// TIA Portal V19 export
FUNCTION_BLOCK "DecoilersHRot_FB"   // FB40, LAD
TITLE = DECOILERS HORIZONTAL ROTATION
// stored: MemoryReserve 100, SetENOAutomatically false
   VAR_INPUT
      AreaInterface : "AreaInterface";
      ZSI : "udt_ZoneSafetyInterface";
      DSI : Struct
         Rotation : "udt_DeviceSafetyInterface";
         Pivot : "udt_DeviceSafetyInterface";
         Translation : "udt_DeviceSafetyInterface";
      END_STRUCT;
      Drive : Struct
         Traslation : "TAx_DriveInterface";
      END_STRUCT;
      HW_ID : Struct
         Traslation_TEL1 : HW_SUBMODULE;
         TraslationEnc_IO : HW_SUBMODULE;
      END_STRUCT;
      DataIn : Struct
         PB_Decoiler1_MoveInLine : Bool;
         PB_Decoiler2_MoveInLine : Bool;
         Rotation : "ValveMachine_DataIn";
         Pivot : "ValveMachine_DataIn";
         Traslation : "Positioning_DOL_Machine_DataIn";
      END_STRUCT;
      CIn : Struct
         Manager : "DecoilersHRot_Manager";
         CoilCar_OutOfLine : Bool;
         PressureRunning_Rotation : Bool;
         PressureRunning_Pivot : Bool;
      END_STRUCT;
      Config : Struct
         Rotation : "ValveMachine_Config";
         Pivot : "ValveMachine_Config";
         Traslation : "Positioning_DOL_Machine_Config";
      END_STRUCT;
   END_VAR
   VAR_OUTPUT
      MachineInterface : "MachineInterface";
      DataOut : Struct
         Rotation : "ValveMachine_DataOut";
         Pivot : "ValveMachine_DataOut";
         Tower_Lamp : Bool;
         Tower_Horn : Bool;
      END_STRUCT;
      COut : "DecoilersHRot_Status";
   END_VAR
   VAR_IN_OUT
      PersistentValues : Struct
         Par : Struct
            TraslationAx : "Positioning_DOL_Machine_Par";
            TraslationEnc : "PosFbk_RTN";
            Traslation_AutSpeed : Real;
         END_STRUCT;
         Ax_Pers : "Positioning_DOL_Machine_Pers_Data";
      END_STRUCT;
   END_VAR
   VAR
      Warning : Struct
         Rotation : "ValveMachine_Wng";
         Pivot : "ValveMachine_Wng";
         Traslation : "Positioning_DOL_Machine_Wng";
         Rotation_NotInPosition : Bool;
         Pivot_NotWork : Bool;
         Translation_NotInPosition : Bool;
      END_STRUCT;
      Alarm : Struct
         Rotation : "ValveAlr";
         Pivot : "ValveAlr";
         Traslation_Ax : "Positioning_DOL_Machine_Alr";
         Traslation_Enc : "PosFbk_Encoder_Alr";
         Rotation_NotInPosition : Bool;
         Pivot_NotWork : Bool;
      END_STRUCT;
      Sts : Struct
         Decoiler1_InLine_Partial : Bool;
         Decoiler2_InLine_Partial : Bool;
      END_STRUCT;
      Ctrl : Struct
         Decoiler1_MoveInLine_Man : Bool;
         Decoiler2_MoveInLine_Man : Bool;
         Decoiler1_MoveInLine_Aut : Bool;
         Decoiler2_MoveInLine_Aut : Bool;
         Decoiler1_MoveInLine : Bool;
         Decoiler2_MoveInLine : Bool;
      END_STRUCT;
      Rotation : "ValveMachine_FB";
      Pivot : "ValveMachine_FB";
      Translation : "Positioning_DOL_Machine_FB";
      Traslation_Enc : "PosFbk_SickAFM60";
      Traslation_EncITF : "PosFbk_ITF";
      TON_Rotation_NotInPosition : TON_TIME;
      TON_Pivot_NotWork : TON_TIME;
      TON_Translation_NotInPosition { S7_SetPoint := 'True'} : TON_TIME;
      AUX : Struct
         Move_Pb_InLineDecoiler1 : Bool;
         Move_Pb_InLineDecoiler2 : Bool;
      END_STRUCT;
   END_VAR
   VAR_TEMP
      Decoiler_N : Int;
      Target : LReal;
      InPosition : Bool;
   END_VAR
   VAR_TEMP   // added for the SCL form of the ladder/FBD networks
      _w1 : Bool;
      _w2 : Bool;
      _w3 : Bool;
   END_VAR
BEGIN

REGION Network 1: Man move in line
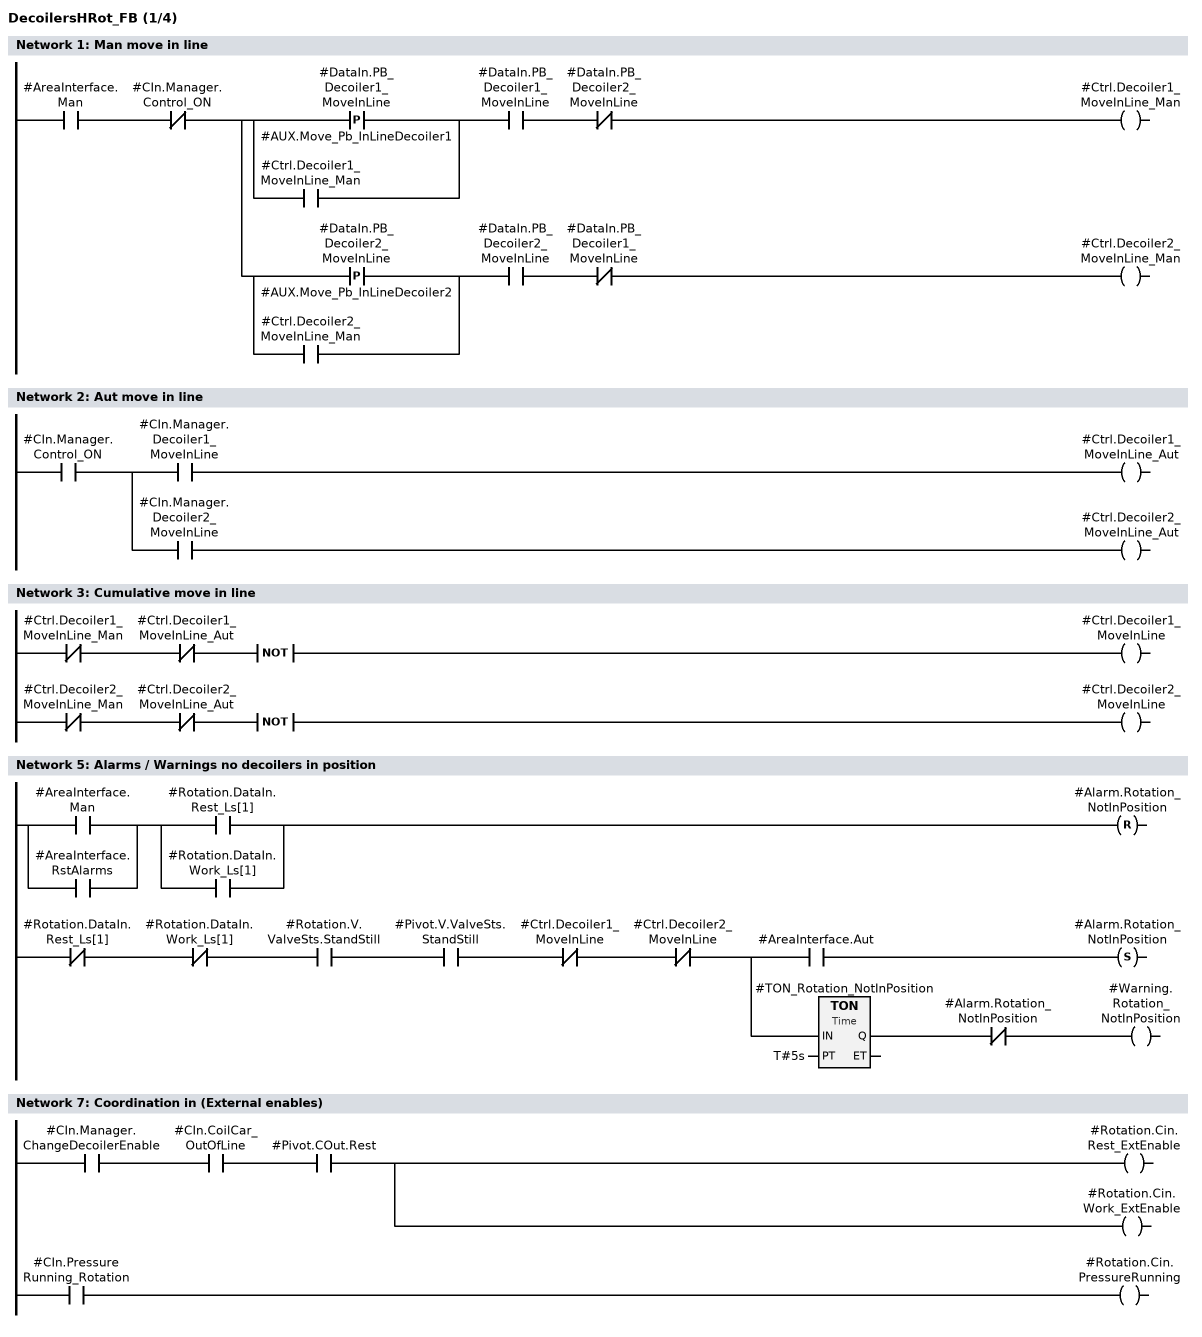
   RUNG wire#powerrail
      Contact( #AreaInterface.Man )
      I_Contact( #CIn.Manager.Control_ON )
      wire#w1
      P_Contact(operand := #DataIn.PB_Decoiler1_MoveInLine, bit := #AUX.Move_Pb_InLineDecoiler1)
      wire#w2
      Contact( #DataIn.PB_Decoiler1_MoveInLine )
      I_Contact( #DataIn.PB_Decoiler2_MoveInLine )
      Coil( #Ctrl.Decoiler1_MoveInLine_Man )
   END_RUNG
   RUNG wire#w1
      Contact( #Ctrl.Decoiler1_MoveInLine_Man )
   END_RUNG wire#w2
   RUNG wire#w1
      P_Contact(operand := #DataIn.PB_Decoiler2_MoveInLine, bit := #AUX.Move_Pb_InLineDecoiler2)
      wire#w3
      Contact( #DataIn.PB_Decoiler2_MoveInLine )
      I_Contact( #DataIn.PB_Decoiler1_MoveInLine )
      Coil( #Ctrl.Decoiler2_MoveInLine_Man )
   END_RUNG
   RUNG wire#w1
      Contact( #Ctrl.Decoiler2_MoveInLine_Man )
   END_RUNG wire#w3
   // the same network as SCL:
   #_w1 := #AreaInterface.Man AND NOT #CIn.Manager.Control_ON;
   #_w2 := #_w1 AND #DataIn.PB_Decoiler1_MoveInLine AND NOT #AUX.Move_Pb_InLineDecoiler1;   // rising edge of #DataIn.PB_Decoiler1_MoveInLine
   #AUX.Move_Pb_InLineDecoiler1 := #DataIn.PB_Decoiler1_MoveInLine;
   #Ctrl.Decoiler1_MoveInLine_Man := (#_w2 OR (#_w1 AND #Ctrl.Decoiler1_MoveInLine_Man)) AND #DataIn.PB_Decoiler1_MoveInLine AND NOT #DataIn.PB_Decoiler2_MoveInLine;
   #_w3 := #_w1 AND #DataIn.PB_Decoiler2_MoveInLine AND NOT #AUX.Move_Pb_InLineDecoiler2;   // rising edge of #DataIn.PB_Decoiler2_MoveInLine
   #AUX.Move_Pb_InLineDecoiler2 := #DataIn.PB_Decoiler2_MoveInLine;
   #Ctrl.Decoiler2_MoveInLine_Man := (#_w3 OR (#_w1 AND #Ctrl.Decoiler2_MoveInLine_Man)) AND #DataIn.PB_Decoiler2_MoveInLine AND NOT #DataIn.PB_Decoiler1_MoveInLine;
END_REGION

REGION Network 2: Aut move in line
   RUNG wire#powerrail
      Contact( #CIn.Manager.Control_ON )
      wire#w1
      Contact( #CIn.Manager.Decoiler1_MoveInLine )
      Coil( #Ctrl.Decoiler1_MoveInLine_Aut )
   END_RUNG
   RUNG wire#w1
      Contact( #CIn.Manager.Decoiler2_MoveInLine )
      Coil( #Ctrl.Decoiler2_MoveInLine_Aut )
   END_RUNG
   // the same network as SCL:
   #Ctrl.Decoiler1_MoveInLine_Aut := #CIn.Manager.Control_ON AND #CIn.Manager.Decoiler1_MoveInLine;
   #Ctrl.Decoiler2_MoveInLine_Aut := #CIn.Manager.Control_ON AND #CIn.Manager.Decoiler2_MoveInLine;
END_REGION

REGION Network 3: Cumulative move in line
   RUNG wire#powerrail
      I_Contact( #Ctrl.Decoiler1_MoveInLine_Man )
      I_Contact( #Ctrl.Decoiler1_MoveInLine_Aut )
      Not()
      Coil( #Ctrl.Decoiler1_MoveInLine )
   END_RUNG
   RUNG wire#powerrail
      I_Contact( #Ctrl.Decoiler2_MoveInLine_Man )
      I_Contact( #Ctrl.Decoiler2_MoveInLine_Aut )
      Not()
      Coil( #Ctrl.Decoiler2_MoveInLine )
   END_RUNG
   // the same network as SCL:
   #Ctrl.Decoiler1_MoveInLine := NOT (NOT #Ctrl.Decoiler1_MoveInLine_Man AND NOT #Ctrl.Decoiler1_MoveInLine_Aut);
   #Ctrl.Decoiler2_MoveInLine := NOT (NOT #Ctrl.Decoiler2_MoveInLine_Man AND NOT #Ctrl.Decoiler2_MoveInLine_Aut);
END_REGION

REGION Network 4: <<< ROTATION >>
END_REGION

REGION Network 5: Alarms / Warnings no decoilers in position
   RUNG wire#powerrail
      Contact( #AreaInterface.Man )
      wire#w1
      Contact( #Rotation.DataIn.Rest_Ls[1] )
      wire#w2
      R_Coil( #Alarm.Rotation_NotInPosition )
   END_RUNG
   RUNG wire#powerrail
      Contact( #AreaInterface.RstAlarms )
   END_RUNG wire#w1
   RUNG wire#w1
      Contact( #Rotation.DataIn.Work_Ls[1] )
   END_RUNG wire#w2
   RUNG wire#powerrail
      I_Contact( #Rotation.DataIn.Rest_Ls[1] )
      I_Contact( #Rotation.DataIn.Work_Ls[1] )
      Contact( #Rotation.V.ValveSts.StandStill )
      Contact( #Pivot.V.ValveSts.StandStill )
      I_Contact( #Ctrl.Decoiler1_MoveInLine )
      I_Contact( #Ctrl.Decoiler2_MoveInLine )
      wire#w3
      Contact( #AreaInterface.Aut )
      S_Coil( #Alarm.Rotation_NotInPosition )
   END_RUNG
   RUNG wire#w3
      { S7_Templates := "time_type := Time" } #TON_Rotation_NotInPosition.TON(pt := T#5s, et =>)
      I_Contact( #Alarm.Rotation_NotInPosition )
      Coil( #Warning.Rotation_NotInPosition )
   END_RUNG
   // the same network as SCL:
   IF (#AreaInterface.Man OR #AreaInterface.RstAlarms) AND (#Rotation.DataIn.Rest_Ls[1] OR #Rotation.DataIn.Work_Ls[1]) THEN
       #Alarm.Rotation_NotInPosition := FALSE;
   END_IF;
   #_w1 := NOT #Rotation.DataIn.Rest_Ls[1] AND NOT #Rotation.DataIn.Work_Ls[1] AND #Rotation.V.ValveSts.StandStill AND #Pivot.V.ValveSts.StandStill AND NOT #Ctrl.Decoiler1_MoveInLine AND NOT #Ctrl.Decoiler2_MoveInLine;
   IF #_w1 AND #AreaInterface.Aut THEN #Alarm.Rotation_NotInPosition := TRUE; END_IF;
   #TON_Rotation_NotInPosition(IN := #_w1, PT := T#5s);   // TON
   #Warning.Rotation_NotInPosition := #TON_Rotation_NotInPosition.Q AND NOT #Alarm.Rotation_NotInPosition;
END_REGION

REGION Network 6 (SCL): Coordination in (Manager)
   #Rotation.Cin.Manager.EnableStopDoorOpeningReq := #CIn.Manager.EnableStopDoorOpeningReq;
   #Rotation.Cin.Manager.EnableStopInPhase := #CIn.Manager.EnableStopInPhase;
   #Rotation.Cin.Manager.EnableStopProgrammed := #CIn.Manager.EnableStopProgrammed;

   // Rotazione @Rest = Decoiler 1 in linea
   // Rotazione @Work = Decoiler 2 in linea

   #Rotation.Cin.Manager.Rest := NOT #Rotation.COut.Rest AND #Ctrl.Decoiler1_MoveInLine;

   #Rotation.Cin.Manager.Work :=  NOT #Rotation.COut.Work AND #Ctrl.Decoiler2_MoveInLine;


   #Rotation.Cin.Manager.Control_ON := #CIn.Manager.Control_ON OR #Rotation.Cin.Manager.Rest OR #Rotation.Cin.Manager.Work;
END_REGION

REGION Network 7: Coordination in (External enables)
   RUNG wire#powerrail
      Contact( #CIn.Manager.ChangeDecoilerEnable )
      Contact( #CIn.CoilCar_OutOfLine )
      Contact( #Pivot.COut.Rest )
      wire#w1
      Coil( #Rotation.Cin.Rest_ExtEnable )
   END_RUNG
   RUNG wire#w1
      Coil( #Rotation.Cin.Work_ExtEnable )
   END_RUNG
   RUNG wire#powerrail
      Contact( #CIn.PressureRunning_Rotation )
      Coil( #Rotation.Cin.PressureRunning )
   END_RUNG
   // the same network as SCL:
   #Rotation.Cin.Rest_ExtEnable := #CIn.Manager.ChangeDecoilerEnable AND #CIn.CoilCar_OutOfLine AND #Pivot.COut.Rest;
   #Rotation.Cin.Work_ExtEnable := #Rotation.Cin.Rest_ExtEnable;
   #Rotation.Cin.PressureRunning := #CIn.PressureRunning_Rotation;
END_REGION

REGION Network 8: External alrms used only for cycle aborting
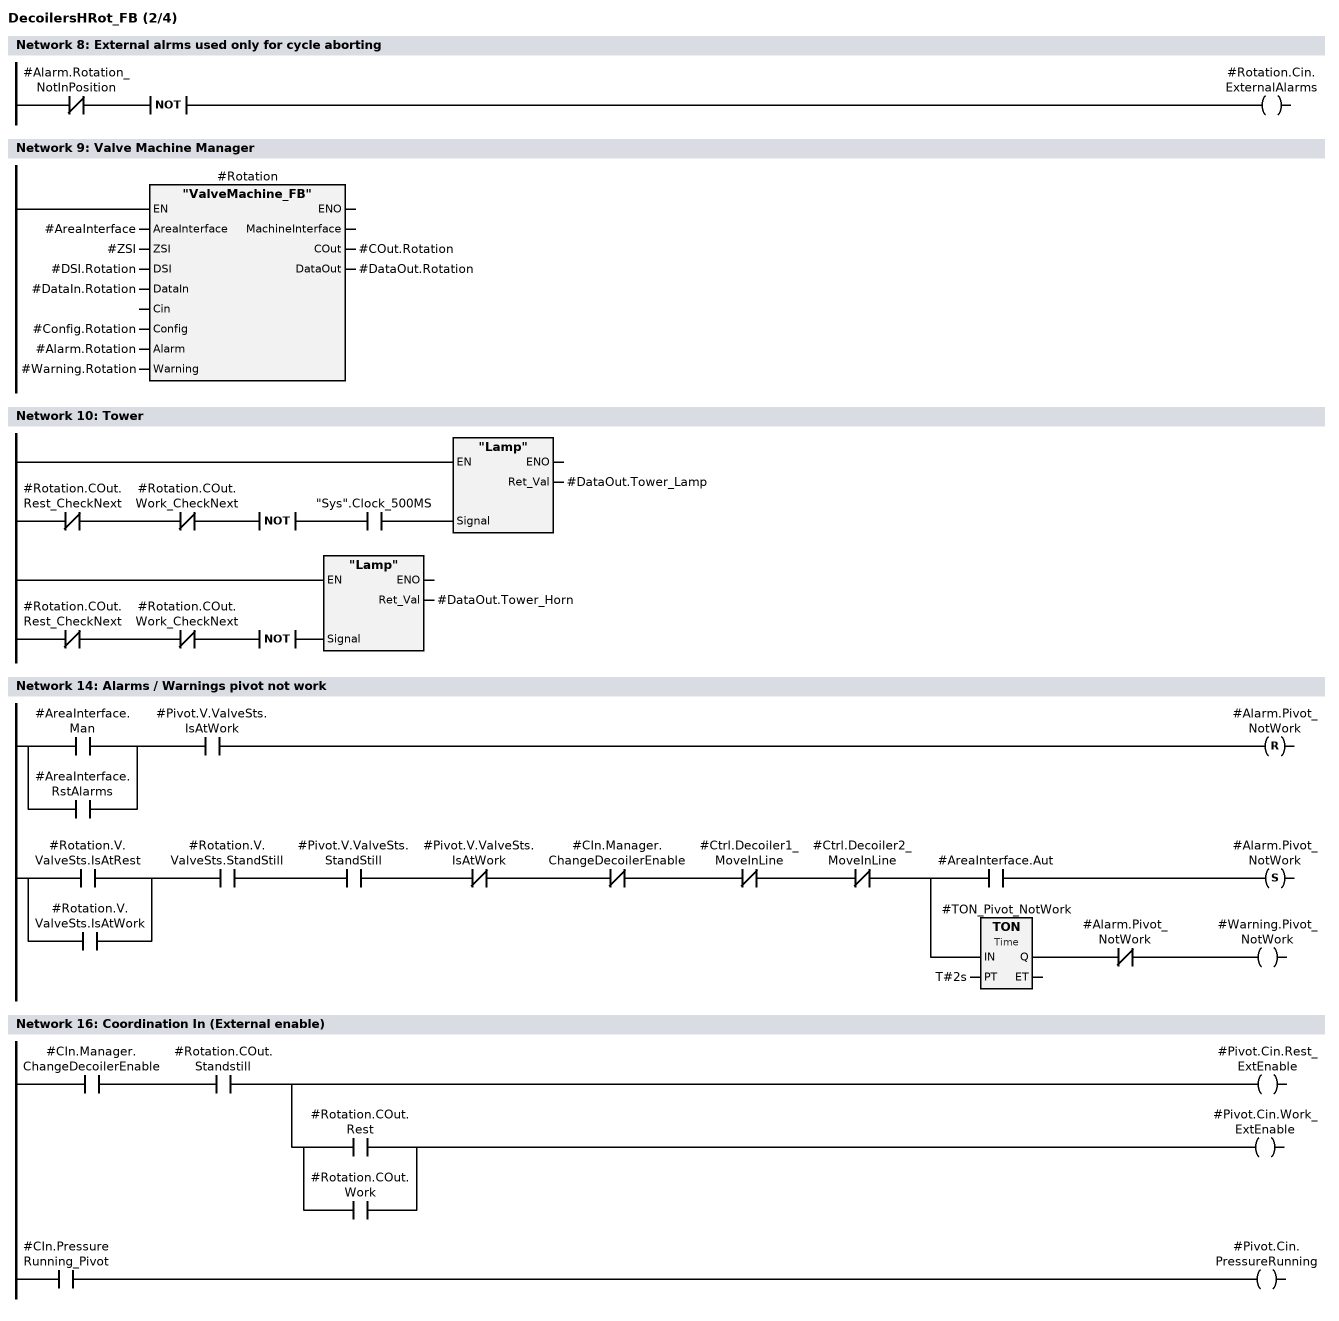
   RUNG wire#powerrail
      I_Contact( #Alarm.Rotation_NotInPosition )
      Not()
      Coil( #Rotation.Cin.ExternalAlarms )
   END_RUNG
   // the same network as SCL:
   #Rotation.Cin.ExternalAlarms := NOT (NOT #Alarm.Rotation_NotInPosition);
END_REGION

REGION Network 9: Valve Machine Manager
   RUNG wire#powerrail
      #Rotation(AreaInterface := #AreaInterface, ZSI := #ZSI, DSI := #DSI.Rotation, DataIn := #DataIn.Rotation, Cin :=, Config := #Config.Rotation, Alarm := #Alarm.Rotation, Warning := #Warning.Rotation, MachineInterface =>, COut => #COut.Rotation, DataOut => #DataOut.Rotation)
   END_RUNG
   // the same network as SCL:
   #Rotation(AreaInterface := #AreaInterface,   // "ValveMachine_FB"
             ZSI := #ZSI,
             DSI := #DSI.Rotation,
             DataIn := #DataIn.Rotation,
             Config := #Config.Rotation,
             Alarm := #Alarm.Rotation,
             Warning := #Warning.Rotation,
             COut => #COut.Rotation,
             DataOut => #DataOut.Rotation);
END_REGION

REGION Network 10: Tower
   RUNG wire#powerrail
      "Lamp"(Signal := wire#w1, Ret_Val => #DataOut.Tower_Lamp)
   END_RUNG
   RUNG wire#powerrail
      I_Contact( #Rotation.COut.Rest_CheckNext )
      I_Contact( #Rotation.COut.Work_CheckNext )
      Not()
      Contact( "Sys".Clock_500MS )
   END_RUNG wire#w1
   RUNG wire#powerrail
      "Lamp"(Signal := wire#w2, Ret_Val => #DataOut.Tower_Horn)
   END_RUNG
   RUNG wire#powerrail
      I_Contact( #Rotation.COut.Rest_CheckNext )
      I_Contact( #Rotation.COut.Work_CheckNext )
      Not()
   END_RUNG wire#w2
   // the same network as SCL:
   #DataOut.Tower_Lamp := "Lamp"(Signal := NOT (NOT #Rotation.COut.Rest_CheckNext AND NOT #Rotation.COut.Work_CheckNext) AND "Sys".Clock_500MS);
   #DataOut.Tower_Horn := "Lamp"(Signal := NOT (NOT #Rotation.COut.Rest_CheckNext AND NOT #Rotation.COut.Work_CheckNext));
END_REGION

REGION Network 11: >
END_REGION

REGION Network 12: >
END_REGION

REGION Network 13: <<< PIVOT >>
END_REGION

REGION Network 14: Alarms / Warnings pivot not work
   RUNG wire#powerrail
      Contact( #AreaInterface.Man )
      wire#w1
      Contact( #Pivot.V.ValveSts.IsAtWork )
      R_Coil( #Alarm.Pivot_NotWork )
   END_RUNG
   RUNG wire#powerrail
      Contact( #AreaInterface.RstAlarms )
   END_RUNG wire#w1
   RUNG wire#powerrail
      Contact( #Rotation.V.ValveSts.IsAtRest )
      wire#w2
      Contact( #Rotation.V.ValveSts.StandStill )
      Contact( #Pivot.V.ValveSts.StandStill )
      I_Contact( #Pivot.V.ValveSts.IsAtWork )
      I_Contact( #CIn.Manager.ChangeDecoilerEnable )
      I_Contact( #Ctrl.Decoiler1_MoveInLine )
      I_Contact( #Ctrl.Decoiler2_MoveInLine )
      wire#w3
      Contact( #AreaInterface.Aut )
      S_Coil( #Alarm.Pivot_NotWork )
   END_RUNG
   RUNG wire#powerrail
      Contact( #Rotation.V.ValveSts.IsAtWork )
   END_RUNG wire#w2
   RUNG wire#w3
      { S7_Templates := "time_type := Time" } #TON_Pivot_NotWork.TON(pt := T#2s, et =>)
      I_Contact( #Alarm.Pivot_NotWork )
      Coil( #Warning.Pivot_NotWork )
   END_RUNG
   // the same network as SCL:
   IF (#AreaInterface.Man OR #AreaInterface.RstAlarms) AND #Pivot.V.ValveSts.IsAtWork THEN
       #Alarm.Pivot_NotWork := FALSE;
   END_IF;
   #_w1 := (#Rotation.V.ValveSts.IsAtRest OR #Rotation.V.ValveSts.IsAtWork) AND #Rotation.V.ValveSts.StandStill AND #Pivot.V.ValveSts.StandStill AND NOT #Pivot.V.ValveSts.IsAtWork AND NOT #CIn.Manager.ChangeDecoilerEnable AND NOT #Ctrl.Decoiler1_MoveInLine AND NOT #Ctrl.Decoiler2_MoveInLine;
   IF #_w1 AND #AreaInterface.Aut THEN #Alarm.Pivot_NotWork := TRUE; END_IF;
   #TON_Pivot_NotWork(IN := #_w1, PT := T#2s);   // TON
   #Warning.Pivot_NotWork := #TON_Pivot_NotWork.Q AND NOT #Alarm.Pivot_NotWork;
END_REGION

REGION Network 15 (SCL): Coordination in (Manager)
   #Pivot.Cin.Manager.EnableStopDoorOpeningReq := #CIn.Manager.EnableStopDoorOpeningReq;
   #Pivot.Cin.Manager.EnableStopInPhase := #CIn.Manager.EnableStopInPhase;
   #Pivot.Cin.Manager.EnableStopProgrammed := #CIn.Manager.EnableStopProgrammed;


   // Rotazione @Rest = Decoiler 1 in linea
   // Rotazione @Work = Decoiler 2 in linea


   #Pivot.Cin.Manager.Rest :=
   (
   (#Ctrl.Decoiler1_MoveInLine AND NOT #Rotation.COut.Rest)
   OR
   (#Ctrl.Decoiler2_MoveInLine AND NOT #Rotation.COut.Work)
   );

   #Pivot.Cin.Manager.Work :=
   NOT #Pivot.Cin.Manager.Rest
   AND
   (
   #Ctrl.Decoiler1_MoveInLine
   OR
   #Ctrl.Decoiler2_MoveInLine);


   #Pivot.Cin.Manager.Control_ON := #CIn.Manager.Control_ON OR #Pivot.Cin.Manager.Work OR #Pivot.Cin.Manager.Rest;
END_REGION

REGION Network 16: Coordination In (External enable)
   RUNG wire#powerrail
      Contact( #CIn.Manager.ChangeDecoilerEnable )
      Contact( #Rotation.COut.Standstill )
      wire#w1
      Coil( #Pivot.Cin.Rest_ExtEnable )
   END_RUNG
   RUNG wire#w1
      Contact( #Rotation.COut.Rest )
      wire#w2
      Coil( #Pivot.Cin.Work_ExtEnable )
   END_RUNG
   RUNG wire#w1
      Contact( #Rotation.COut.Work )
   END_RUNG wire#w2
   RUNG wire#powerrail
      Contact( #CIn.PressureRunning_Pivot )
      Coil( #Pivot.Cin.PressureRunning )
   END_RUNG
   // the same network as SCL:
   #Pivot.Cin.Rest_ExtEnable := #CIn.Manager.ChangeDecoilerEnable AND #Rotation.COut.Standstill;
   #Pivot.Cin.Work_ExtEnable := #Pivot.Cin.Rest_ExtEnable AND (#Rotation.COut.Rest OR #Rotation.COut.Work);
   #Pivot.Cin.PressureRunning := #CIn.PressureRunning_Pivot;
END_REGION

REGION Network 17: External alrms used only for cycle aborting
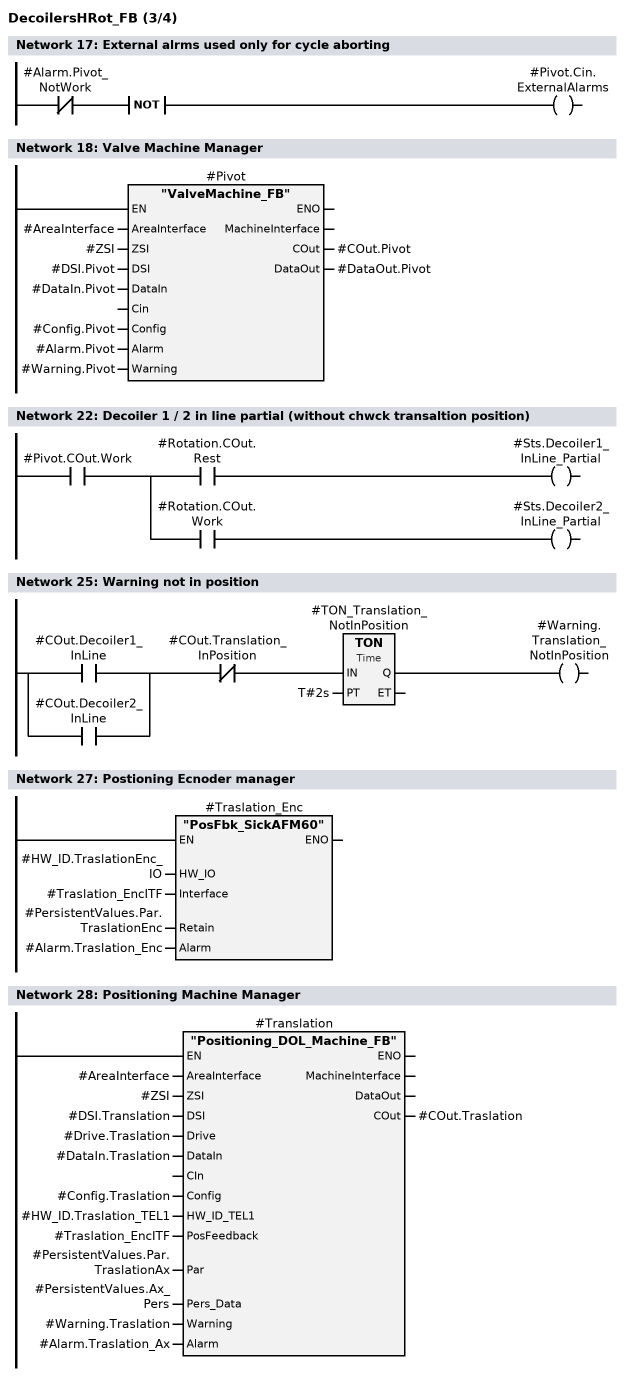
   RUNG wire#powerrail
      I_Contact( #Alarm.Pivot_NotWork )
      Not()
      Coil( #Pivot.Cin.ExternalAlarms )
   END_RUNG
   // the same network as SCL:
   #Pivot.Cin.ExternalAlarms := NOT (NOT #Alarm.Pivot_NotWork);
END_REGION

REGION Network 18: Valve Machine Manager
   RUNG wire#powerrail
      #Pivot(AreaInterface := #AreaInterface, ZSI := #ZSI, DSI := #DSI.Pivot, DataIn := #DataIn.Pivot, Cin :=, Config := #Config.Pivot, Alarm := #Alarm.Pivot, Warning := #Warning.Pivot, MachineInterface =>, COut => #COut.Pivot, DataOut => #DataOut.Pivot)
   END_RUNG
   // the same network as SCL:
   #Pivot(AreaInterface := #AreaInterface,   // "ValveMachine_FB"
          ZSI := #ZSI,
          DSI := #DSI.Pivot,
          DataIn := #DataIn.Pivot,
          Config := #Config.Pivot,
          Alarm := #Alarm.Pivot,
          Warning := #Warning.Pivot,
          COut => #COut.Pivot,
          DataOut => #DataOut.Pivot);
END_REGION

REGION Network 19: >
END_REGION

REGION Network 20: >
END_REGION

REGION Network 22: Decoiler 1 / 2 in line partial (without chwck transaltion position)
   RUNG wire#powerrail
      Contact( #Pivot.COut.Work )
      wire#w1
      Contact( #Rotation.COut.Rest )
      Coil( #Sts.Decoiler1_InLine_Partial )
   END_RUNG
   RUNG wire#w1
      Contact( #Rotation.COut.Work )
      Coil( #Sts.Decoiler2_InLine_Partial )
   END_RUNG
   // the same network as SCL:
   #Sts.Decoiler1_InLine_Partial := #Pivot.COut.Work AND #Rotation.COut.Rest;
   #Sts.Decoiler2_InLine_Partial := #Pivot.COut.Work AND #Rotation.COut.Work;
END_REGION

REGION Network 23: <<< TRASLATION >>
END_REGION

REGION Network 24 (SCL): Coordination In (Manager)



   // Gestione comandi manager
   // 
   #Translation.CIn.Manager.EnableStopDoorOpeningReq := #CIn.Manager.EnableStopDoorOpeningReq;
   #Translation.CIn.Manager.EnableStopInPhase := #CIn.Manager.EnableStopInPhase;
   #Translation.CIn.Manager.EnableStopProgrammed := #CIn.Manager.EnableStopProgrammed;


   #Translation.CIn.Manager.Minus := FALSE;
   #Translation.CIn.Manager.Plus := FALSE;

   #Translation.CIn.Manager.MoveToPos := #Ctrl.Decoiler1_MoveInLine OR #Ctrl.Decoiler2_MoveInLine;

   #Translation.CIn.Manager.Control_ON := #CIn.Manager.Control_ON OR #Translation.CIn.Manager.MoveToPos;


   #Translation.CIn.Manager.Speed := #PersistentValues.Par.TraslationAx.Man_Speed;


   // Posizione desiderta / comandata





   IF #Ctrl.Decoiler1_MoveInLine
       OR
       (NOT #Ctrl.Decoiler1_MoveInLine_Man AND NOT #Ctrl.Decoiler2_MoveInLine_Man AND #Sts.Decoiler1_InLine_Partial)
   THEN
       #Decoiler_N := 1;
   END_IF;

   IF #Ctrl.Decoiler2_MoveInLine
       OR
       (NOT #Ctrl.Decoiler1_MoveInLine_Man AND NOT #Ctrl.Decoiler2_MoveInLine_Man AND #Sts.Decoiler2_InLine_Partial)
   THEN
       #Decoiler_N := 2;
   END_IF;

   #Translation.CIn.Manager.Pos :=
   "DecHRot_Calc_Translation_By_MaterialWidth"(Decoiler_N := #Decoiler_N,
                                               Material_Width :="PPrf_MAIN".ON_WORK.GeneralData.Material_Width);
END_REGION

REGION Network 25: Warning not in position
   RUNG wire#powerrail
      Contact( #COut.Decoiler1_InLine )
      wire#w1
      I_Contact( #COut.Translation_InPosition )
      { S7_Templates := "time_type := Time" } #TON_Translation_NotInPosition.TON(pt := T#2s, et =>)
      Coil( #Warning.Translation_NotInPosition )
   END_RUNG
   RUNG wire#powerrail
      Contact( #COut.Decoiler2_InLine )
   END_RUNG wire#w1
   // the same network as SCL:
   #TON_Translation_NotInPosition(IN := (#COut.Decoiler1_InLine OR #COut.Decoiler2_InLine) AND NOT #COut.Translation_InPosition,   // TON
                           PT := T#2s);
   #Warning.Translation_NotInPosition := #TON_Translation_NotInPosition.Q;
END_REGION

REGION Network 26 (SCL): Coordination In (External enable + External alarm + Position limits)
   #Translation.CIn.MinusExtEnable := #CIn.CoilCar_OutOfLine;

   #Translation.CIn.PlusExtEnable := #CIn.CoilCar_OutOfLine;

   #Translation.CIn.ExternalAlarms := FALSE;


   #Translation.CIn.PositionLimits.EnableMin := FALSE;
   #Translation.CIn.PositionLimits.EnableMax := FALSE;
END_REGION

REGION Network 27: Postioning Ecnoder manager
   RUNG wire#powerrail
      #Traslation_Enc(HW_IO := #HW_ID.TraslationEnc_IO, Interface := #Traslation_EncITF, Retain := #PersistentValues.Par.TraslationEnc, Alarm := #Alarm.Traslation_Enc)
   END_RUNG
   // the same network as SCL:
   #Traslation_Enc(HW_IO := #HW_ID.TraslationEnc_IO,   // "PosFbk_SickAFM60"
                   Interface := #Traslation_EncITF,
                   Retain := #PersistentValues.Par.TraslationEnc,
                   Alarm := #Alarm.Traslation_Enc);
END_REGION

REGION Network 28: Positioning Machine Manager
   RUNG wire#powerrail
      #Translation(AreaInterface := #AreaInterface, ZSI := #ZSI, DSI := #DSI.Translation, Drive := #Drive.Traslation, DataIn := #DataIn.Traslation, CIn :=, Config := #Config.Traslation, HW_ID_TEL1 := #HW_ID.Traslation_TEL1, PosFeedback := #Traslation_EncITF, Par := #PersistentValues.Par.TraslationAx, Pers_Data := #PersistentValues.Ax_Pers, Warning := #Warning.Traslation, Alarm := #Alarm.Traslation_Ax, MachineInterface =>, DataOut =>, COut => #COut.Traslation)
   END_RUNG
   // the same network as SCL:
   #Translation(AreaInterface := #AreaInterface,   // "Positioning_DOL_Machine_FB"
                ZSI := #ZSI,
                DSI := #DSI.Translation,
                Drive := #Drive.Traslation,
                DataIn := #DataIn.Traslation,
                Config := #Config.Traslation,
                HW_ID_TEL1 := #HW_ID.Traslation_TEL1,
                PosFeedback := #Traslation_EncITF,
                Par := #PersistentValues.Par.TraslationAx,
                Pers_Data := #PersistentValues.Ax_Pers,
                Warning := #Warning.Traslation,
                Alarm := #Alarm.Traslation_Ax,
                COut => #COut.Traslation);
END_REGION

REGION Network 29: >
END_REGION

REGION Network 30: >
END_REGION

REGION Network 31: <<< MACHINE STATUS >>>
END_REGION

REGION Network 32: Machine coordination out
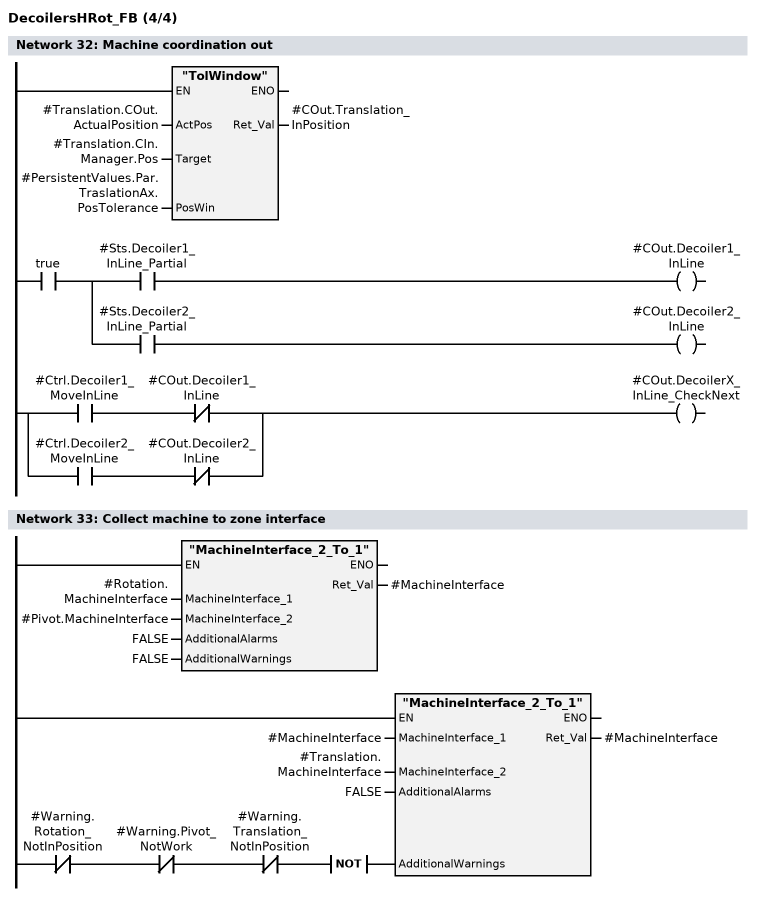
   RUNG wire#powerrail
      "TolWindow"(ActPos := #Translation.COut.ActualPosition, Target := #Translation.CIn.Manager.Pos, PosWin := #PersistentValues.Par.TraslationAx.PosTolerance, Ret_Val => #COut.Translation_InPosition)
   END_RUNG
   RUNG wire#powerrail
      Contact( true )
      wire#w1
      Contact( #Sts.Decoiler1_InLine_Partial )
      Coil( #COut.Decoiler1_InLine )
   END_RUNG
   RUNG wire#w1
      Contact( #Sts.Decoiler2_InLine_Partial )
      Coil( #COut.Decoiler2_InLine )
   END_RUNG
   RUNG wire#powerrail
      Contact( #Ctrl.Decoiler1_MoveInLine )
      I_Contact( #COut.Decoiler1_InLine )
      wire#w2
      Coil( #COut.DecoilerX_InLine_CheckNext )
   END_RUNG
   RUNG wire#powerrail
      Contact( #Ctrl.Decoiler2_MoveInLine )
      I_Contact( #COut.Decoiler2_InLine )
   END_RUNG wire#w2
   // the same network as SCL:
   #COut.Translation_InPosition := "TolWindow"(ActPos := #Translation.COut.ActualPosition,
                           Target := #Translation.CIn.Manager.Pos,
                           PosWin := #PersistentValues.Par.TraslationAx.PosTolerance);
   #COut.Decoiler1_InLine := true AND #Sts.Decoiler1_InLine_Partial;
   #COut.Decoiler2_InLine := true AND #Sts.Decoiler2_InLine_Partial;
   #COut.DecoilerX_InLine_CheckNext := (#Ctrl.Decoiler1_MoveInLine AND NOT #COut.Decoiler1_InLine) OR (#Ctrl.Decoiler2_MoveInLine AND NOT #COut.Decoiler2_InLine);
END_REGION

REGION Network 33: Collect machine to zone interface
   RUNG wire#powerrail
      "MachineInterface_2_To_1"(MachineInterface_1 := #Rotation.MachineInterface, MachineInterface_2 := #Pivot.MachineInterface, AdditionalAlarms := FALSE, AdditionalWarnings := FALSE, Ret_Val => #MachineInterface)
   END_RUNG
   RUNG wire#powerrail
      "MachineInterface_2_To_1"(AdditionalWarnings := wire#w1, MachineInterface_1 := #MachineInterface, MachineInterface_2 := #Translation.MachineInterface, AdditionalAlarms := FALSE, Ret_Val => #MachineInterface)
   END_RUNG
   RUNG wire#powerrail
      I_Contact( #Warning.Rotation_NotInPosition )
      I_Contact( #Warning.Pivot_NotWork )
      I_Contact( #Warning.Translation_NotInPosition )
      Not()
   END_RUNG wire#w1
   // the same network as SCL:
   #MachineInterface := "MachineInterface_2_To_1"(MachineInterface_1 := #Rotation.MachineInterface,
                           MachineInterface_2 := #Pivot.MachineInterface,
                           AdditionalAlarms := FALSE,
                           AdditionalWarnings := FALSE);
   #MachineInterface := "MachineInterface_2_To_1"(MachineInterface_1 := #MachineInterface,
                           MachineInterface_2 := #Translation.MachineInterface,
                           AdditionalAlarms := FALSE,
                           AdditionalWarnings := NOT (NOT #Warning.Rotation_NotInPosition AND NOT #Warning.Pivot_NotWork AND NOT #Warning.Translation_NotInPosition));
END_REGION

REGION Network 34: >
END_REGION

REGION Network 35: >
END_REGION

REGION Network 36: >
END_REGION
END_FUNCTION_BLOCK
